// TIA Portal V17 export
// export: Created 2024-09-02T12:49:53.9539558Z, ExportSetting WithDefaults, DisplayName Totally Integrated Automation Portal, DisplayVersion V17, DisplayName TIA Portal Openness, DisplayVersion V17, DisplayName TIA Portal Version Control Interface, DisplayVersion V17, DisplayName STEP 7 Professional, DisplayVersion V17, DisplayName STEP 7 Safety, DisplayVersion V17, DisplayName WinCC Professional, DisplayVersion V17
FUNCTION "AnwFC_Safety_Connect" : Void   // FC7001, LAD
TITLE = Transfer signals to F program / Signale an F-Programm übergeben
{ S7_Optimized_Access := 'TRUE' }
AUTHOR : OlegFuehrus
FAMILY : Safe
NAME : Safe
VERSION : 0.1
// Used to ensure data consistency Changes in the standard program therefore have no influence on the safety program. The controller does not have to be in STOP mode to load the standard program.
// Dient zur Absicherung der Datenkonsitenz
// Änderungen im Standardprogramm haben dadurch keinen Einfluss auf das
// Sicherheitsprogramm. Die Steuerung muss auch nicht im Betriebszustand
// STOP sein, um das Standardprogramm zu laden.
// stored: AutoNumber false, IsIECCheckEnabled false, SetENOAutomatically false, UDAEnableTagReadback false
   VAR_TEMP
      t_numof_opened_door : Int;   // Anzahl der offenen Schutztüren / Number of open safety doors
      t_numof_E22 : Int;   // Anzahl der betätigten E22-Schliessungen / Number of actuated E22 locks
   END_VAR
BEGIN

REGION Network 1: F-Program - Media On / an F-Programm - Medien Ein
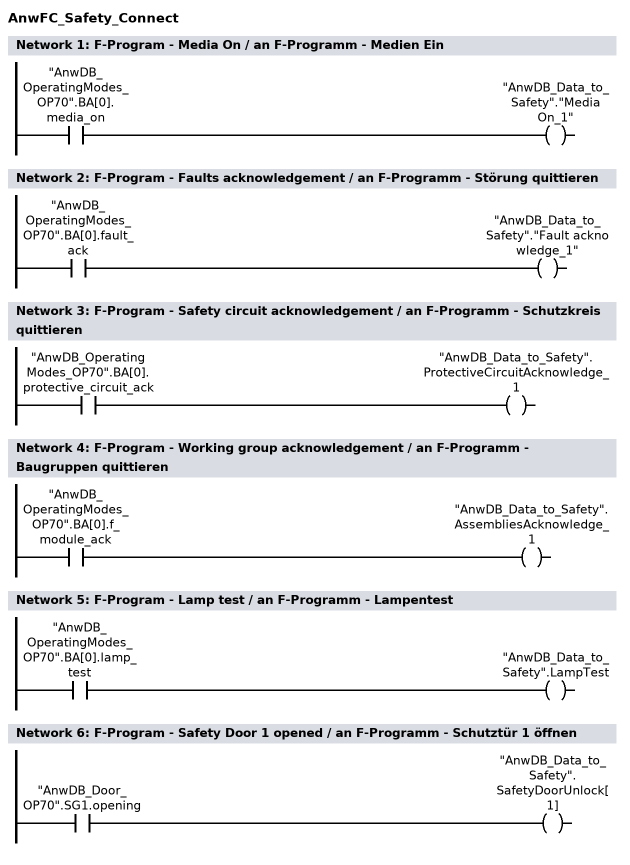
   RUNG wire#powerrail
      Contact( "AnwDB_OperatingModes_OP70".BA[0].media_on )
      Coil( "AnwDB_Data_to_Safety"."Media On_1" )
   END_RUNG
   // the same network as SCL:
   "AnwDB_Data_to_Safety"."Media On_1" := "AnwDB_OperatingModes_OP70".BA[0].media_on;
END_REGION

REGION Network 2: F-Program - Faults acknowledgement / an F-Programm - Störung quittieren
   RUNG wire#powerrail
      Contact( "AnwDB_OperatingModes_OP70".BA[0].fault_ack )
      Coil( "AnwDB_Data_to_Safety"."Fault acknowledge_1" )
   END_RUNG
   // the same network as SCL:
   "AnwDB_Data_to_Safety"."Fault acknowledge_1" := "AnwDB_OperatingModes_OP70".BA[0].fault_ack;
END_REGION

REGION Network 3: F-Program - Safety circuit acknowledgement / an F-Programm - Schutzkreis quittieren
   RUNG wire#powerrail
      Contact( "AnwDB_OperatingModes_OP70".BA[0].protective_circuit_ack )
      Coil( "AnwDB_Data_to_Safety".ProtectiveCircuitAcknowledge_1 )
   END_RUNG
   // the same network as SCL:
   "AnwDB_Data_to_Safety".ProtectiveCircuitAcknowledge_1 := "AnwDB_OperatingModes_OP70".BA[0].protective_circuit_ack;
END_REGION

REGION Network 4: F-Program - Working group acknowledgement / an F-Programm - Baugruppen quittieren
   RUNG wire#powerrail
      Contact( "AnwDB_OperatingModes_OP70".BA[0].f_module_ack )
      Coil( "AnwDB_Data_to_Safety".AssembliesAcknowledge_1 )
   END_RUNG
   // the same network as SCL:
   "AnwDB_Data_to_Safety".AssembliesAcknowledge_1 := "AnwDB_OperatingModes_OP70".BA[0].f_module_ack;
END_REGION

REGION Network 5: F-Program - Lamp test / an F-Programm - Lampentest
   RUNG wire#powerrail
      Contact( "AnwDB_OperatingModes_OP70".BA[0].lamp_test )
      Coil( "AnwDB_Data_to_Safety".LampTest )
   END_RUNG
   // the same network as SCL:
   "AnwDB_Data_to_Safety".LampTest := "AnwDB_OperatingModes_OP70".BA[0].lamp_test;
END_REGION

REGION Network 6: F-Program - Safety Door 1 opened / an F-Programm - Schutztür 1 öffnen
   RUNG wire#powerrail
      Contact( "AnwDB_Door_OP70".SG1.opening )
      Coil( "AnwDB_Data_to_Safety".SafetyDoorUnlock[1] )
   END_RUNG
   // the same network as SCL:
   "AnwDB_Data_to_Safety".SafetyDoorUnlock[1] := "AnwDB_Door_OP70".SG1.opening;
END_REGION
END_FUNCTION
